ADAPTER IEmergencySludgeBuffer (* Adapter Interface *)
  (* Standard: 61499-1 *)
  (* Version 0.0, 9/17/2026, Schneider Electric *)
  PACKAGE SE.Nereda;
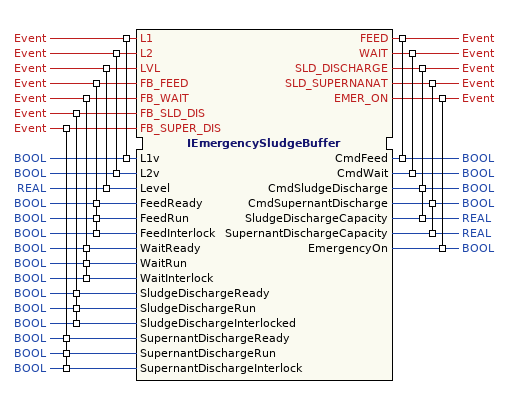
  EVENT_INPUT
    L1 WITH L1v;
    L2 WITH L2v;
    LVL WITH Level;
    FB_FEED WITH FeedReady, FeedRun, FeedInterlock;
    FB_WAIT WITH WaitReady, WaitRun, WaitInterlock;
    FB_SLD_DIS WITH SludgeDischargeReady, SludgeDischargeRun, SludgeDischargeInterlocked;
    FB_SUPER_DIS WITH SupernantDischargeReady, SupernantDischargeRun, SupernantDischargeInterlock;
  END_EVENT
  EVENT_OUTPUT
    FEED WITH CmdFeed;
    WAIT WITH CmdWait;
    SLD_DISCHARGE WITH CmdSludgeDischarge, SludgeDischargeCapacity;
    SLD_SUPERNANAT WITH CmdSupernantDischarge, SupernantDischargeCapacity;
    EMER_ON WITH EmergencyOn;
  END_EVENT
  VAR_INPUT
    L1v : BOOL;
    L2v : BOOL;
    Level : REAL;
    FeedReady : BOOL;
    FeedRun : BOOL;
    FeedInterlock : BOOL;
    WaitReady : BOOL;
    WaitRun : BOOL;
    WaitInterlock : BOOL;
    SludgeDischargeReady : BOOL;
    SludgeDischargeRun : BOOL;
    SludgeDischargeInterlocked : BOOL;
    SupernantDischargeReady : BOOL;
    SupernantDischargeRun : BOOL;
    SupernantDischargeInterlock : BOOL;
  END_VAR
  VAR_OUTPUT
    CmdFeed : BOOL;
    CmdWait : BOOL;
    CmdSludgeDischarge : BOOL;
    CmdSupernantDischarge : BOOL;
    SludgeDischargeCapacity : REAL;
    SupernantDischargeCapacity : REAL;
    EmergencyOn : BOOL;
  END_VAR
  SERVICE SOCKET/PLUG
    SEQUENCE request_confirm
      SOCKET.REQ(REQD) -> PLUG.REQ(REQD);
      PLUG.CNF(CNFD) -> SOCKET.CNF(CNFD);
    END_SEQUENCE
    SEQUENCE indication_response
      PLUG.IND(INDD) -> SOCKET.IND(INDD);
      SOCKET.RSP(RSPD) -> PLUG.RSP(RSPD);
    END_SEQUENCE
  END_SERVICE
END_ADAPTER
